// TIA Portal V20 export
DATA_BLOCK "DB_RealTime"   // DB107
// stored: InstanceOfName FB_RealTime, InstanceOfType FB
"FB_RealTime"
BEGIN
END_DATA_BLOCK
